FUNCTION_BLOCK RenderComp (* Composite Function Block Type *)
  (* Standard: 61499-2 *)
  (* Version 0.2, 2003-12-05, JHC, Rockwell Automation, Renamed from NEWCOMPFB. *)
  (* Version 0.1, 2002-01-08, JHC, Rockwell Automation, Added DLY FB as example. *)
  (* Version 0.0, 2000-05-27, JHC, Rockwell Automation *)
  (* Compiler header: package fb.rt.cs725;import fb.rt.vhmi.*; *)
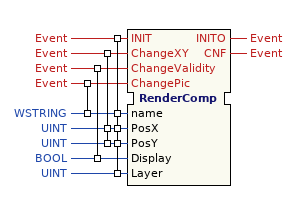
  EVENT_INPUT
    INIT WITH name, PosX, PosY, Layer; (* Initialization Request *)
    ChangeXY WITH PosX, PosY; (* Normal Execution Request *)
    ChangeValidity WITH Display;
    ChangePic WITH name;
  END_EVENT
  EVENT_OUTPUT
    INITO; (* Initialization Confirm *)
    CNF; (* Execution Confirmation *)
  END_EVENT
  VAR_INPUT
    name : WSTRING;
    PosX : UINT;
    PosY : UINT;
    Display : BOOL;
    Layer : UINT;
  END_VAR
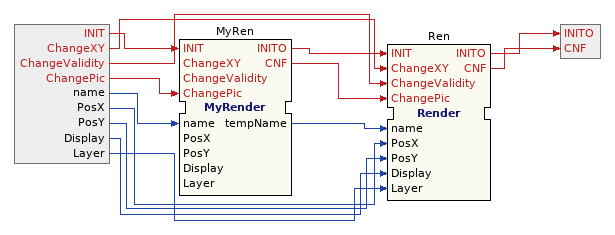
  FBS
    MyRen : MyRender;
    Ren : Render;
  END_FBS
  EVENT_CONNECTIONS
    INIT TO MyRen.INIT;
    MyRen.INITO TO Ren.INIT;
    Ren.INITO TO INITO;
    ChangeXY TO Ren.ChangeXY;
    ChangeValidity TO Ren.ChangeValidity;
    ChangePic TO MyRen.ChangePic;
    MyRen.CNF TO Ren.ChangePic;
    Ren.CNF TO CNF;
  END_CONNECTIONS
  DATA_CONNECTIONS
    MyRen.tempName TO Ren.name;
    name TO MyRen.name;
    PosX TO Ren.PosX;
    PosY TO Ren.PosY;
    Display TO Ren.Display;
    Layer TO Ren.Layer;
  END_CONNECTIONS
END_FUNCTION_BLOCK
